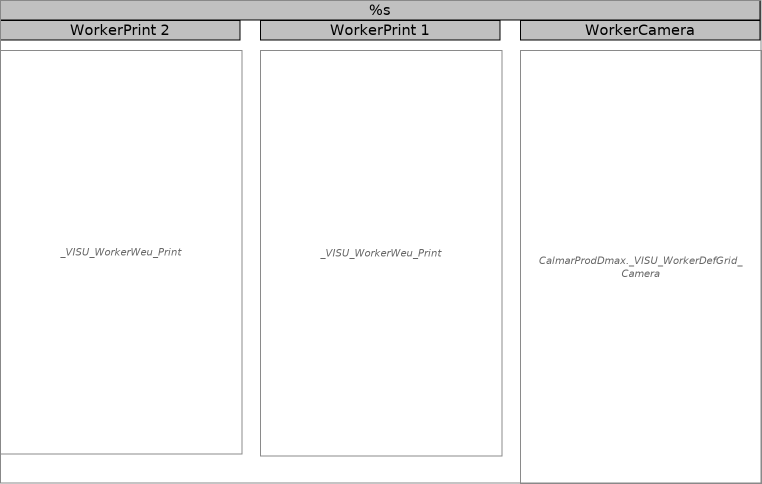
VISUALIZATION _VISU_Worker_Pm  // 762x484
VAR_IN_OUT
	mInst : FB_PrintModule_WEU;
END_VAR
    Frame (0,50 242x404)
        shows _VISU_WorkerWeu_Print(m_Inst := mInst.fbWorkerPrint[2])
    Frame (260,50 242x406)
        shows _VISU_WorkerWeu_Print(m_Inst := mInst.fbWorkerPrint[1])
    Rectangle (0,20 240x20), "WorkerPrint 2"
    Rectangle (260,20 240x20), "WorkerPrint 1"
    Frame (520,50 242x434)
        shows CalmarProdDmax._VISU_WorkerDefGrid_Camera(m_Inst := mInst.fbWorkerCamera)
    Rectangle (520,20 240x20), "WorkerCamera"
    Rectangle (0,0 760x20), "%s", text variable: mInst._pAdsPm^.aO_Name
END_VISUALIZATION

(* stored: Version 1.1.0.1, ProductVersion 3.1.4024.11
   Visu _VISU_Worker_Pm: Id {32d4a689-e6b6-4214-ac3e-087879e7f035} *)
